FUNCTION_BLOCK FB_AdjustLongPress
VAR_INPUT
END_VAR
VAR_OUTPUT
END_VAR
VAR
	m_adjustOnTime :LREAL :=0;
	m_timeThres :LREAL :=2.0;
END_VAR

// check if instrument is on
METHOD run : BOOL
VAR_INPUT
	IOValue :UDINT;
END_VAR
run := m_adjustOnTime>m_timeThres AND 4<>(IOValue AND 10#4);

// adjust io is 3th bit 
IF 4=(IOValue AND 10#4) THEN
	m_adjustOnTime :=m_adjustOnTime+g_slaveArmCtrlCycleTime;
ELSE
	m_adjustOnTime :=0;
END_IF
END_METHOD

END_FUNCTION_BLOCK

(* stored: Version 1.1.0.1, ProductVersion 3.1.4024.11
   POU FB_AdjustLongPress: Id {e0779f91-07c8-4baf-aa2d-030a1a40aeb6}, SpecialFunc None
   Method run: Id {37acad5a-bbd5-4003-a087-e278f155bb55} *)
